(* Logix 5000 project; controller TORQUE Emulate 5570 rev 36.11; software revision 36.00 *)

TASK MainTask (continuous, watchdog 500 ms) : MainProgram, Emulation

MODULES
   Local : Emulate 5570 (ICP 2, rev 36.11)
       : 1756-IB16 (ICP 3, rev 3.1, Input RPI 20 ms)
       : vendor 1 type 7 code 16 (ICP 4, rev 3.1, Output RPI 20 ms)
       : 1756-IF8 (ICP 5, rev 1.1, Input RPI 100 ms)
END_MODULES

VAR_GLOBAL   (* controller tags *)
   AIN_1 : ALIAS FOR Local:5:I.Ch0Data;
   AIN_2 : ALIAS FOR Local:5:I.Ch1Data;
   AIN_3 : ALIAS FOR Local:5:I.Ch2Data;
   AIN_4 : ALIAS FOR Local:5:I.Ch3Data;
   CROSS_THRD_LIMIT : DINT;   // Cross Thread Torque Setting
   CRS_THRD_ERROR : ALIAS FOR Local:4:O.Data.11;   // Cross Thread Indicator
   DN_LS : ALIAS FOR Local:3:I.Data.10;
   DN_SOL : ALIAS FOR Local:4:O.Data.0;
   LOWER_LIMIT : DINT := 95;
   MOTOR_1 : ALIAS FOR Local:4:O.Data.1;
   MOTOR_2 : ALIAS FOR Local:4:O.Data.2;
   MOTOR_3 : ALIAS FOR Local:4:O.Data.3;
   MOTOR_4 : ALIAS FOR Local:4:O.Data.4;
   START_NO_1 : ALIAS FOR Local:3:I.Data.14;
   START_NO_2 : ALIAS FOR Local:3:I.Data.15;
   TO_ERROR : ALIAS FOR Local:4:O.Data.10;
   UPPER_LIMIT : DINT := 100;
END_VAR

PROGRAM Emulation   (* main routine Emulation *)
VAR
   emCROSS_THRD : BOOL;
   emDOWN_SOL_TRAVEL : TIMER := (PRE := 5000);
   emMOTOR1_ONS : BOOL;
   emMOTOR2_ONS : BOOL;
   emMOTOR3_ONS : BOOL;
   emMOTOR4_ONS : BOOL;
   emMOTOR_1_AIN : DINT;
   emMOTOR_1_NO_TORQUE : BOOL;
   emMOTOR_1_OFF_DWELL : TIMER := (PRE := 20);
   emMOTOR_1_ON_DWELL : TIMER := (PRE := 80);
   emMOTOR_2_AIN : DINT;
   emMOTOR_2_ON_DWELL : TIMER := (PRE := 50);
   emMOTOR_3_AIN : DINT;
   emMOTOR_3_ON_DWELL : TIMER := (PRE := 60);
   emMOTOR_4_AIN : DINT;
   emMOTOR_4_CRS_DWELL : TIMER := (PRE := 20);
   emMOTOR_4_ON_DWELL : TIMER := (PRE := 20);
   emNO_TORQUE : BOOL;
   emPART_TRACK : COUNTER := (PRE := 5);
   emSET_POINT : DINT := 97;
END_VAR

ROUTINE Emulation   (* ladder *)
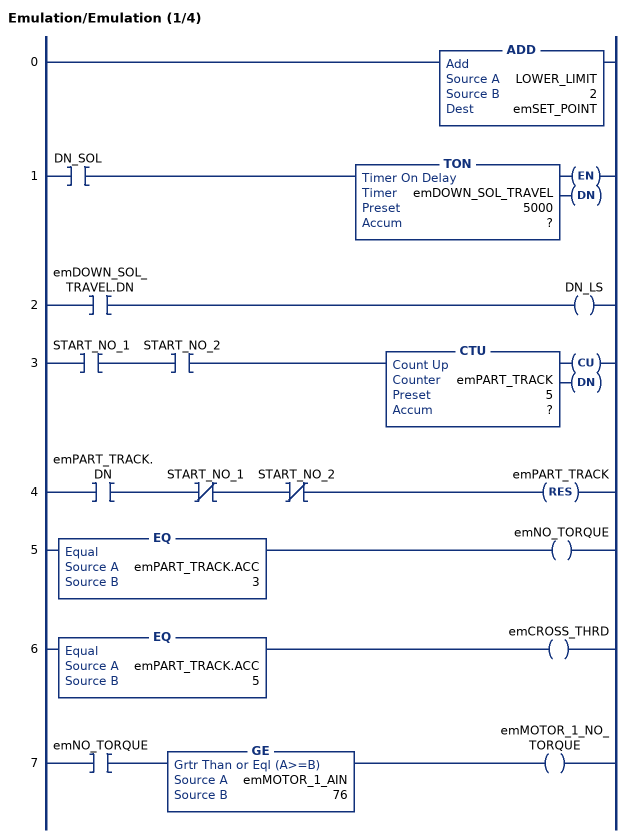
   0: ADD(LOWER_LIMIT,2,emSET_POINT);
   1: XIC(DN_SOL)TON(emDOWN_SOL_TRAVEL,?,?);
   2: XIC(emDOWN_SOL_TRAVEL.DN)OTE(DN_LS);
   3: XIC(START_NO_1)XIC(START_NO_2)CTU(emPART_TRACK,?,?);
   4: XIC(emPART_TRACK.DN)XIO(START_NO_1)XIO(START_NO_2)RES(emPART_TRACK);
   5: EQ(emPART_TRACK.ACC,3)OTE(emNO_TORQUE);
   6: EQ(emPART_TRACK.ACC,5)OTE(emCROSS_THRD);
   7: XIC(emNO_TORQUE)GE(emMOTOR_1_AIN,76)OTE(emMOTOR_1_NO_TORQUE);
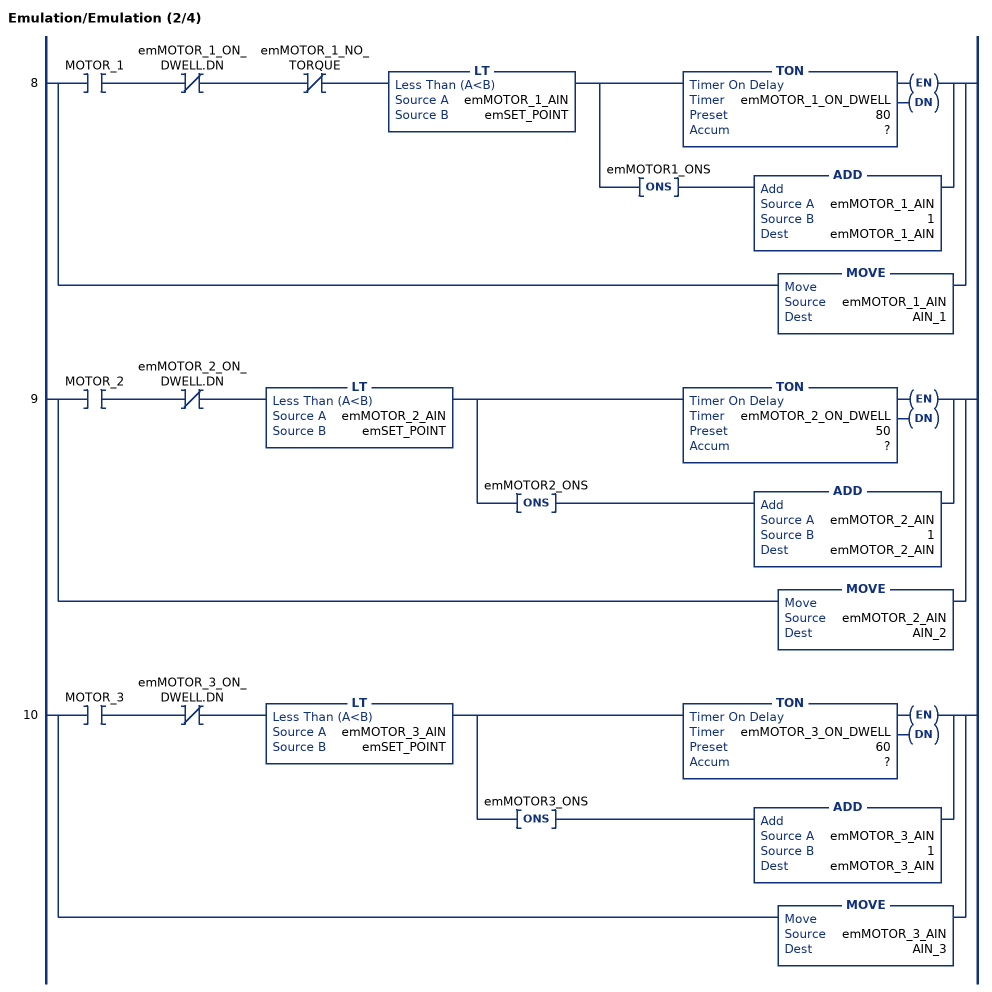
   8: [XIC(MOTOR_1) XIO(emMOTOR_1_ON_DWELL.DN) XIO(emMOTOR_1_NO_TORQUE) LT(emMOTOR_1_AIN,emSET_POINT) [TON(emMOTOR_1_ON_DWELL,?,?) ,ONS(emMOTOR1_ONS) ADD(emMOTOR_1_AIN,1,emMOTOR_1_AIN) ] ,MOVE(emMOTOR_1_AIN,AIN_1) ];
   9: [XIC(MOTOR_2) XIO(emMOTOR_2_ON_DWELL.DN) LT(emMOTOR_2_AIN,emSET_POINT) [TON(emMOTOR_2_ON_DWELL,?,?) ,ONS(emMOTOR2_ONS) ADD(emMOTOR_2_AIN,1,emMOTOR_2_AIN) ] ,MOVE(emMOTOR_2_AIN,AIN_2) ];
   10: [XIC(MOTOR_3) XIO(emMOTOR_3_ON_DWELL.DN) LT(emMOTOR_3_AIN,emSET_POINT) [TON(emMOTOR_3_ON_DWELL,?,?) ,ONS(emMOTOR3_ONS) ADD(emMOTOR_3_AIN,1,emMOTOR_3_AIN) ] ,MOVE(emMOTOR_3_AIN,AIN_3) ];
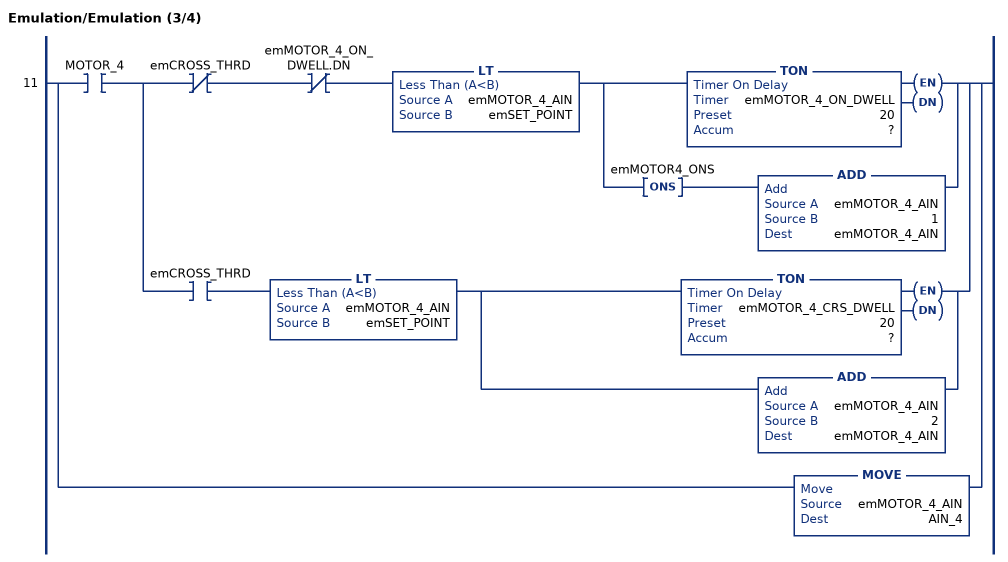
   11: [XIC(MOTOR_4) [XIO(emCROSS_THRD) XIO(emMOTOR_4_ON_DWELL.DN) LT(emMOTOR_4_AIN,emSET_POINT) [TON(emMOTOR_4_ON_DWELL,?,?) ,ONS(emMOTOR4_ONS) ADD(emMOTOR_4_AIN,1,emMOTOR_4_AIN) ] ,XIC(emCROSS_THRD) LT(emMOTOR_4_AIN,emSET_POINT) [TON(emMOTOR_4_CRS_DWELL,?,?) ,ADD(emMOTOR_4_AIN,2,emMOTOR_4_AIN) ] ] ,MOVE(emMOTOR_4_AIN,AIN_4) ];
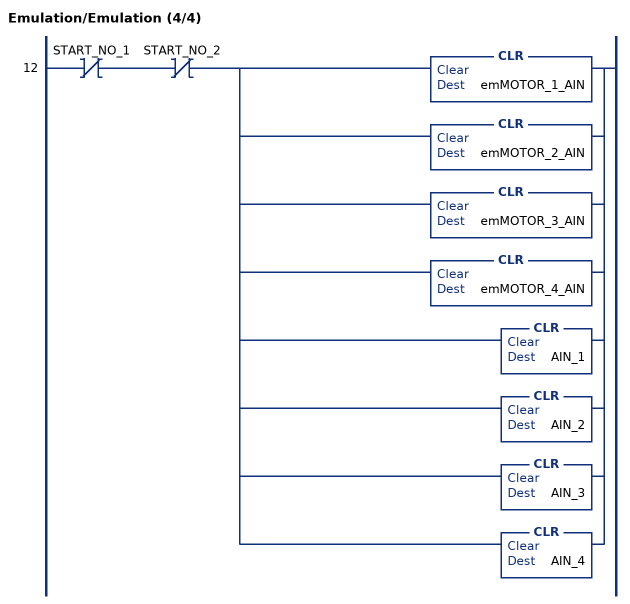
   12: XIO(START_NO_1)XIO(START_NO_2)[CLR(emMOTOR_1_AIN) ,CLR(emMOTOR_2_AIN) ,CLR(emMOTOR_3_AIN) ,CLR(emMOTOR_4_AIN) ,CLR(AIN_1) ,CLR(AIN_2) ,CLR(AIN_3) ,CLR(AIN_4) ];
END_ROUTINE
END_PROGRAM

PROGRAM MainProgram   (* main routine MainRoutine *)
VAR
   CROSS_THRD_1 : BOOL;   // No. 1 Bolt Cross Threaded
   CROSS_THRD_2 : BOOL;   // No. 2 Bolt Cross Threaded
   CROSS_THRD_3 : BOOL;   // No. 3 Bolt Cross Threaded
   CROSS_THRD_4 : BOOL;   // No. 4 Bolt Cross Threaded
   CRS_THRD_DWELL : TIMER := (PRE := 2000);   // Cross Thread DWELL
   TO_DWELL : TIMER := (PRE := 20000);
        .DN   // Time Out Dwell
        .EN   // Time Out Enabled (EN)
        .TT   // Time Out Elapsing (TT) Optional
   TORQUE_1_NOT_SET : BOOL;   // No. 1 Bolt Not at Torque
   TORQUE_1_SET : BOOL;
   TORQUE_2_NOT_SET : BOOL;   // No. 2 Bolt Not At Torque
   TORQUE_2_SET : BOOL;
   TORQUE_3_NOT_SET : BOOL;   // No. 3 Bolt Not at Torque
   TORQUE_3_SET : BOOL;
   TORQUE_4_NOT_SET : BOOL;   // No. 4 Bolt Not At Torque
   TORQUE_4_SET : BOOL;
END_VAR

ROUTINE MainRoutine   (* ladder *)
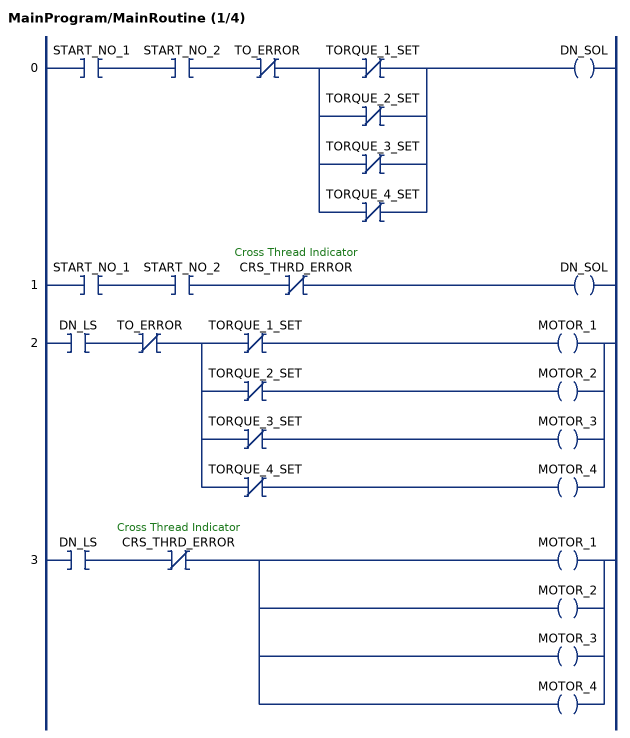
   0: XIC(START_NO_1)XIC(START_NO_2)XIO(TO_ERROR)[XIO(TORQUE_1_SET) ,XIO(TORQUE_2_SET) ,XIO(TORQUE_3_SET) ,XIO(TORQUE_4_SET) ]OTE(DN_SOL);
   1: XIC(START_NO_1)XIC(START_NO_2)XIO(CRS_THRD_ERROR)OTE(DN_SOL);
   2: XIC(DN_LS)XIO(TO_ERROR)[XIO(TORQUE_1_SET) OTE(MOTOR_1) ,XIO(TORQUE_2_SET) OTE(MOTOR_2) ,XIO(TORQUE_3_SET) OTE(MOTOR_3) ,XIO(TORQUE_4_SET) OTE(MOTOR_4) ];
   3: XIC(DN_LS)XIO(CRS_THRD_ERROR)[OTE(MOTOR_1) ,OTE(MOTOR_2) ,OTE(MOTOR_3) ,OTE(MOTOR_4) ];
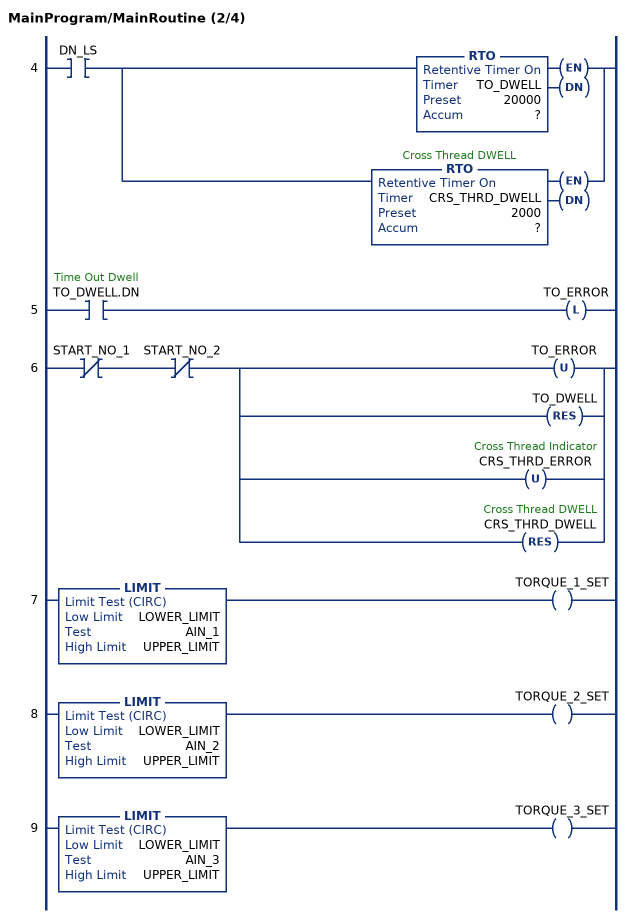
   4: XIC(DN_LS)[RTO(TO_DWELL,?,?) ,RTO(CRS_THRD_DWELL,?,?) ];
   5: XIC(TO_DWELL.DN)OTL(TO_ERROR);
   6: XIO(START_NO_1)XIO(START_NO_2)[OTU(TO_ERROR) ,RES(TO_DWELL) ,OTU(CRS_THRD_ERROR) ,RES(CRS_THRD_DWELL) ];
   7: LIMIT(LOWER_LIMIT,AIN_1,UPPER_LIMIT)OTE(TORQUE_1_SET);
   8: LIMIT(LOWER_LIMIT,AIN_2,UPPER_LIMIT)OTE(TORQUE_2_SET);
   9: LIMIT(LOWER_LIMIT,AIN_3,UPPER_LIMIT)OTE(TORQUE_3_SET);
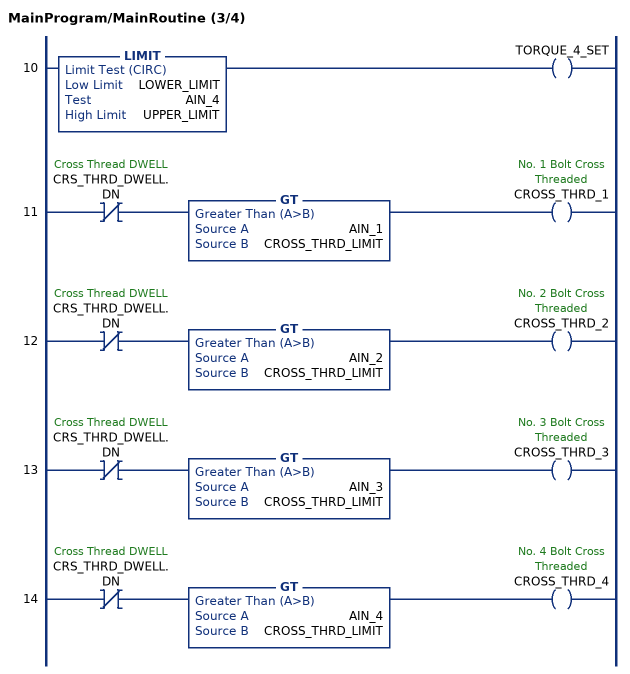
   10: LIMIT(LOWER_LIMIT,AIN_4,UPPER_LIMIT)OTE(TORQUE_4_SET);
   11: XIO(CRS_THRD_DWELL.DN)GT(AIN_1,CROSS_THRD_LIMIT)OTE(CROSS_THRD_1);
   12: XIO(CRS_THRD_DWELL.DN)GT(AIN_2,CROSS_THRD_LIMIT)OTE(CROSS_THRD_2);
   13: XIO(CRS_THRD_DWELL.DN)GT(AIN_3,CROSS_THRD_LIMIT)OTE(CROSS_THRD_3);
   14: XIO(CRS_THRD_DWELL.DN)GT(AIN_4,CROSS_THRD_LIMIT)OTE(CROSS_THRD_4);
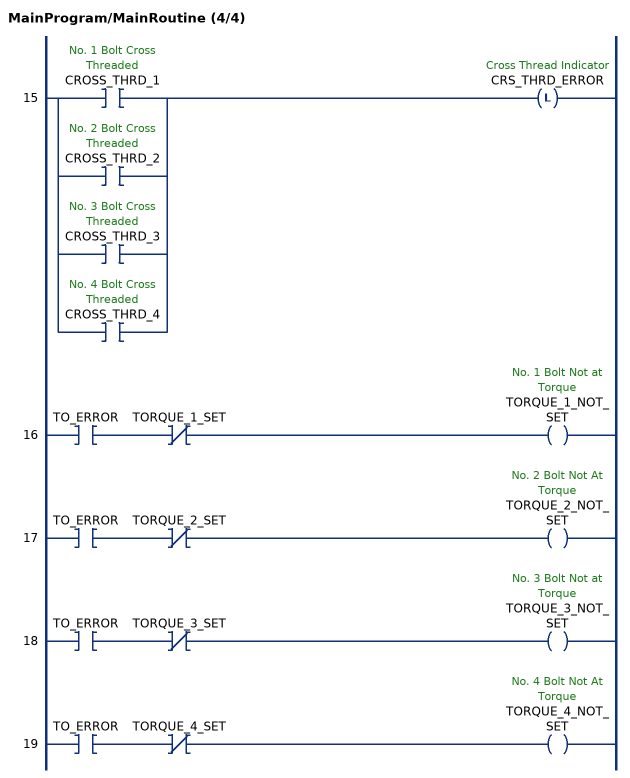
   15: [XIC(CROSS_THRD_1) ,XIC(CROSS_THRD_2) ,XIC(CROSS_THRD_3) ,XIC(CROSS_THRD_4) ]OTL(CRS_THRD_ERROR);
   16: XIC(TO_ERROR)XIO(TORQUE_1_SET)OTE(TORQUE_1_NOT_SET);
   17: XIC(TO_ERROR)XIO(TORQUE_2_SET)OTE(TORQUE_2_NOT_SET);
   18: XIC(TO_ERROR)XIO(TORQUE_3_SET)OTE(TORQUE_3_NOT_SET);
   19: XIC(TO_ERROR)XIO(TORQUE_4_SET)OTE(TORQUE_4_NOT_SET);
END_ROUTINE
END_PROGRAM
